PROGRAM AXIS
VAR
	Axis1: AXIS_REF;
	Axis2: AXIS_REF;
	Axis3: AXIS_REF;
	Axis4: AXIS_REF;
	Axis5: AXIS_REF;
	Axis6: AXIS_REF;
END_VAR

Axis1(
	PlcToNc:= , 
	NcToPlc=> , 
	ADS=> , 
	Status=> , 
	DriveAddress:= );
	
Axis2(
	PlcToNc:= , 
	NcToPlc=> , 
	ADS=> , 
	Status=> , 
	DriveAddress:= );
	
Axis3(
	PlcToNc:= , 
	NcToPlc=> , 
	ADS=> , 
	Status=> , 
	DriveAddress:= );
	
Axis4(
	PlcToNc:= , 
	NcToPlc=> , 
	ADS=> , 
	Status=> , 
	DriveAddress:= );

Axis5(
	PlcToNc:= , 
	NcToPlc=> , 
	ADS=> , 
	Status=> , 
	DriveAddress:= );
	
Axis6(
	PlcToNc:= , 
	NcToPlc=> , 
	ADS=> , 
	Status=> , 
	DriveAddress:= );

END_PROGRAM

(* stored: Version 1.1.0.1, ProductVersion 3.1.4024.0
   POU AXIS: Id {8315ae65-fa76-455a-aa9a-9aba0bcc348d}, SpecialFunc None *)
